FUNCTION_BLOCK ELLIPTICENVELOPE
  {SET_ATTRIBUTE(OpcUa, SERVICE)}
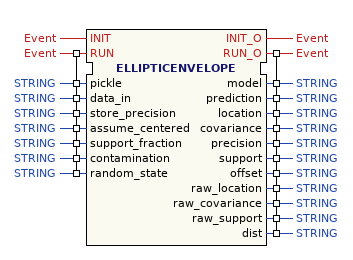
  EVENT_INPUT
    INIT;
    RUN WITH pickle, data_in, store_precision, assume_centered, support_fraction, contamination, random_state; {SET_ATTRIBUTE(OpcUa, Method)}
  END_EVENT
  EVENT_OUTPUT
    INIT_O;
    RUN_O WITH model, prediction, location, covariance, precision, support, offset, raw_location, raw_covariance, raw_support, dist;
  END_EVENT
  VAR_INPUT
    pickle : STRING; {SET_ATTRIBUTE(OpcUa, Variable)}
    data_in : STRING; {SET_ATTRIBUTE(OpcUa, Variable)}
    store_precision : STRING; {SET_ATTRIBUTE(OpcUa, Constant)}
    assume_centered : STRING; {SET_ATTRIBUTE(OpcUa, Constant)}
    support_fraction : STRING; {SET_ATTRIBUTE(OpcUa, Constant)}
    contamination : STRING; {SET_ATTRIBUTE(OpcUa, Constant)}
    random_state : STRING; {SET_ATTRIBUTE(OpcUa, Constant)}
  END_VAR
  VAR_OUTPUT
    model : STRING; {SET_ATTRIBUTE(OpcUa, Variable)}
    prediction : STRING; {SET_ATTRIBUTE(OpcUa, Variable)}
    location : STRING; {SET_ATTRIBUTE(OpcUa, Variable)}
    covariance : STRING; {SET_ATTRIBUTE(OpcUa, Variable)}
    precision : STRING; {SET_ATTRIBUTE(OpcUa, Variable)}
    support : STRING; {SET_ATTRIBUTE(OpcUa, Variable)}
    offset : STRING; {SET_ATTRIBUTE(OpcUa, Variable)}
    raw_location : STRING; {SET_ATTRIBUTE(OpcUa, Variable)}
    raw_covariance : STRING; {SET_ATTRIBUTE(OpcUa, Variable)}
    raw_support : STRING; {SET_ATTRIBUTE(OpcUa, Variable)}
    dist : STRING; {SET_ATTRIBUTE(OpcUa, Variable)}
  END_VAR
END_FUNCTION_BLOCK
